{attribute 'GeneratedUsingTerminal: EL6201-0000-0017'}
{attribute addProperty BoxType "EL6201-0000-0017"}
{attribute addProperty Id "Slave_26A_DI0BOOL1Slave_26A_DI1BOOL1Slave_26A_DI2BOOL1Slave_26A_DI3BOOL1Slave_26B_DI0BOOL1Slave_26B_DI1BOOL1Slave_26B_DI2BOOL1Slave_26B_DI3BOOL1"}
{attribute addProperty CRC "1999433096"}
{attribute addProperty Size "8"}
TYPE Slave_26_Inputs_772CED88 :
STRUCT
	{attribute addProperty Name "Slave_26A_DI0"}
	Slave_26A_DI0 : BOOL;
	{attribute addProperty Name "Slave_26A_DI1"}
	Slave_26A_DI1 : BOOL;
	{attribute addProperty Name "Slave_26A_DI2"}
	Slave_26A_DI2 : BOOL;
	{attribute addProperty Name "Slave_26A_DI3"}
	Slave_26A_DI3 : BOOL;
	{attribute addProperty Name "Slave_26B_DI0"}
	Slave_26B_DI0 : BOOL;
	{attribute addProperty Name "Slave_26B_DI1"}
	Slave_26B_DI1 : BOOL;
	{attribute addProperty Name "Slave_26B_DI2"}
	Slave_26B_DI2 : BOOL;
	{attribute addProperty Name "Slave_26B_DI3"}
	Slave_26B_DI3 : BOOL;
END_STRUCT
END_TYPE

(* stored: Version 1.2.0.0, ProductVersion 3.1.4024.9
   DUT Slave_26_Inputs_772CED88: Id {343e7789-f85b-4f75-b946-fce14826d4dd} *)
